// TwinCAT 3 PLC project PLC
// ProgramVersion: 3.1.4024.0
// libraries:
//   Tc2_Standard, * (Beckhoff Automation GmbH)
//   Tc2_System, * (Beckhoff Automation GmbH)
//   Tc3_Module, * (Beckhoff Automation GmbH)
//   VisuSymbols,3.5.10.0,System
// project tree:
//   Counters/ FB2_Counters.TcPOU
//   / GlobalTextList.TcGTLO, GVL.TcGVL, PlcTask.TcTTO, Visualization Manager.TcVMO (not stored)
//   Interface/ DB10_Alias.TcGVL, DIDO.TcGVL, FC10_Alias.TcPOU
//   Main Functie/ DB_PRG1.TcGVL, FC_PRG1.TcPOU
//   POUs/ FC3_Safety.TcPOU, FC_Comms1.TcPOU, FC_Comms2.TcPOU, FC_StartStopReset.TcPOU, MAIN.TcPOU
//   VISUs/ HMI.TcVIS
// real-time tasks:
//   TASK PlcTask: cycle T#10ms, priority 20, ADS port 350
// I/O:
//   DEVICE EC_Master (EtherCAT), AmsNetId 10.10.10.3.2.1
//     Term 1 (EK1100) [EK1100 EtherCAT Coupler (2A E-Bus)]
//       Term 2 (EL1008) [EL1008 8Ch. Dig. Input 24V, 3ms]
//       Term 3 (EL1008) [EL1008 8Ch. Dig. Input 24V, 3ms]
//       Term 4 (EL2004) [EL2004 4Ch. Dig. Output 24V, 0.5A]
//       Term 5 (EL2004) [EL2004 4Ch. Dig. Output 24V, 0.5A]
//       Term 6 (EL2004) [EL2004 4Ch. Dig. Output 24V, 0.5A]
//       Term 7 (EL9011) [EL9011 End Terminal]
// variable links:
//   PLC/PLC Instance <-> EC_Master (EtherCAT)/Term 1 (EK1100)/Term 2 (EL1008)
//     PlcTask Inputs/DIDO.Ingang{1..8} <-> Channel {1..8}/Input  (8 links)
//   PLC/PLC Instance <-> EC_Master (EtherCAT)/Term 1 (EK1100)/Term 3 (EL1008)
//     PlcTask Inputs/DIDO.Ingang{9..16} <-> Channel {1..8}/Input  (8 links)
//   PLC/PLC Instance <-> EC_Master (EtherCAT)/Term 1 (EK1100)/Term 4 (EL2004)
//     PlcTask Outputs/DIDO.Uitgang{1..4} <-> Channel {1..4}/Output  (4 links)
//   PLC/PLC Instance <-> EC_Master (EtherCAT)/Term 1 (EK1100)/Term 5 (EL2004)
//     PlcTask Outputs/DIDO.Uitgang{5..8} <-> Channel {1..4}/Output  (4 links)
//   PLC/PLC Instance <-> EC_Master (EtherCAT)/Term 1 (EK1100)/Term 6 (EL2004)
//     PlcTask Outputs/DIDO.Uitgang{9..12} <-> Channel {1..4}/Output  (4 links)

CONFIGURATION PLC
    RESOURCE PLC ON TwinCAT3
        TASK PlcTask(INTERVAL := T#10ms, PRIORITY := 20);
        PROGRAM MAIN WITH PlcTask : MAIN;
    END_RESOURCE
END_CONFIGURATION

// ---- GVL.TcGVL
{attribute 'qualified_only'}
VAR_GLOBAL
	
	safetyOK : BOOL := FALSE;
	b_StartPRG : BOOL;
	b_StopPRG : BOOL;
	// KUKA communicaties	
	i_KUKAStatus : INT;
	b_startBeweging : BOOL;
END_VAR

// ---- Interface/DB10_Alias.TcGVL
{attribute 'qualified_only'}
VAR_GLOBAL
		

	b_IOSimulatie : BOOL := FALSE;
	// ingangen Nood, start & stop
	ix_E_stopNC : BOOL;
	ix_startKnop : BOOL;
	ix_stopKnop : BOOL; 
	
	// ingangen fotocel
	ix_lengteFC : BOOL;
	ix_hamsterGripperDetectieFC : BOOL;
	
	ix_reedCuttingtoolCilinderOpen : BOOL;
	ix_reedCuttingtoolCilinderGesloten : BOOL;
	ix_reedGripperCilinder1 : BOOL;
	ix_reedGripperCilinder2 : BOOL;
	
	// start/ stop uitgangen extruder&cutting tool
	qx_relaisExtruderStart : BOOL;
	qx_relaisExtruderStop: BOOL;
	qx_relaisCuttingtoolActiveer : BOOL;
	qx_relaisCuttingtoolDeactiveer : BOOL;
	
	// uitgangen ventielaansturing
	qx_ventielEen : BOOL; 
	qx_ventielTwee : BOOL; 
	
	//uitgangen gereserveerd voor KUKA/Engel communicatie
	// E stop
	// bitlevel comm's
	qx_kukaCommEstop : BOOL; 	// E_stop
	qx_kukaCommStart : BOOL; 		// startcommando
	ix_kukaGereed : BOOL; 		// Gereed/persencompleet
	ix_kukaAlarmIN : BOOL; 		// alarm
	
	
END_VAR

// ---- Interface/DIDO.TcGVL
{attribute 'qualified_only'}
VAR_GLOBAL
	

	// Digitale ingangen
	Ingang1 AT %IX40.0 : BOOL;
	Ingang2 AT %IX40.1 : BOOL;
	Ingang3 AT %IX40.2 : BOOL;
	Ingang4 AT %IX40.3 : BOOL;
	Ingang5 AT %IX40.4 : BOOL;
	Ingang6 AT %IX40.5 : BOOL;
	Ingang7 AT %IX40.6 : BOOL;
	Ingang8 AT %IX40.7 : BOOL;

	Ingang9 AT %IX41.0 : BOOL;
	Ingang10 AT %IX41.1 : BOOL;
	Ingang11 AT %IX41.2 : BOOL;
	Ingang12 AT %IX41.3 : BOOL;
	Ingang13 AT %IX41.4 : BOOL;
	Ingang14 AT %IX41.5 : BOOL;
	Ingang15 AT %IX41.6 : BOOL;
	Ingang16 AT %IX41.7 : BOOL;
	
	
	// Digitale uitgangen
	Uitgang1 AT %QX26.0 : BOOL;
	Uitgang2 AT %QX26.1 : BOOL;
	Uitgang3 AT %QX26.2 : BOOL;
	Uitgang4 AT %QX26.3 : BOOL;
	Uitgang5 AT %QX26.4 : BOOL;
	Uitgang6 AT %QX26.5 : BOOL;
	Uitgang7 AT %QX26.6 : BOOL;
	Uitgang8 AT %QX26.7 : BOOL;
	Uitgang9 AT %QX27.0 : BOOL;
	Uitgang10 AT %QX27.1 : BOOL;
	Uitgang11 AT %QX27.2 : BOOL;
	Uitgang12 AT %QX27.3 : BOOL;	
	
END_VAR

// ---- Main Functie/DB_PRG1.TcGVL
{attribute 'qualified_only'}
VAR_GLOBAL
	PRG1Stap : INT;
	
	t_prgT1_extruderRelaisAan : TON;
	t_prgT2_extruderRelaisStop : TON;
	t_prgT3_cuttingRelaisAan : TON;
	t_prgT4_cuttingRelaisUit : TON;
	t_prgT5_resetKukaGereed : TON; // <<<<<<<<<<<<<<<<< Ter simulatie. IRL signaal van KUKA die dit regelt.
	t_prgT6_Stap60advance : TON;
	t_prgT7_PRGStopRelaisTimer : TON;
	t_prgT8 : TON;
END_VAR

// ---- POUs/MAIN.TcPOU
PROGRAM MAIN
VAR
	FB2_Counters : FB2_Counters;

END_VAR

// Init spulletjes

FB2_Counters();
FC10_Alias();

GVL.safetyOK := FC3_Safety();

// FC Comms from KUKA.
GVL.i_KUKAStatus := FC_Comms1(DB10_Alias.ix_kukaGereed,DB10_Alias.ix_kukaAlarmIN);

FC_StartStopReset();

FC_PRG1(GVL.safetyOK, GVL.i_KUKAStatus); // hardcoded '1' vanaf de KUKA; // GVL.i_KUKAStatus

// FC COmms to KUKA
	
FC_Comms2(GVL.safetyOK,GVL.b_startBeweging);

END_PROGRAM

// ---- Counters/FB2_Counters.TcPOU
FUNCTION_BLOCK FB2_Counters
VAR_INPUT
END_VAR
VAR_OUTPUT
END_VAR
VAR
	t_timerHigh : TON;
	t_timerLow : TP;
	b_eenHzClk : BOOL;
	b_eenHzTrigger : R_Trig;
	i_productieTimerSec: DINT;
	i_productieTimerMin: DINT;
	i_productieTimerHour: DINT;
END_VAR
VAR // added by the converter: edge detectors and wires of the graphical bodies
    _w1, _w2 : BOOL;
END_VAR

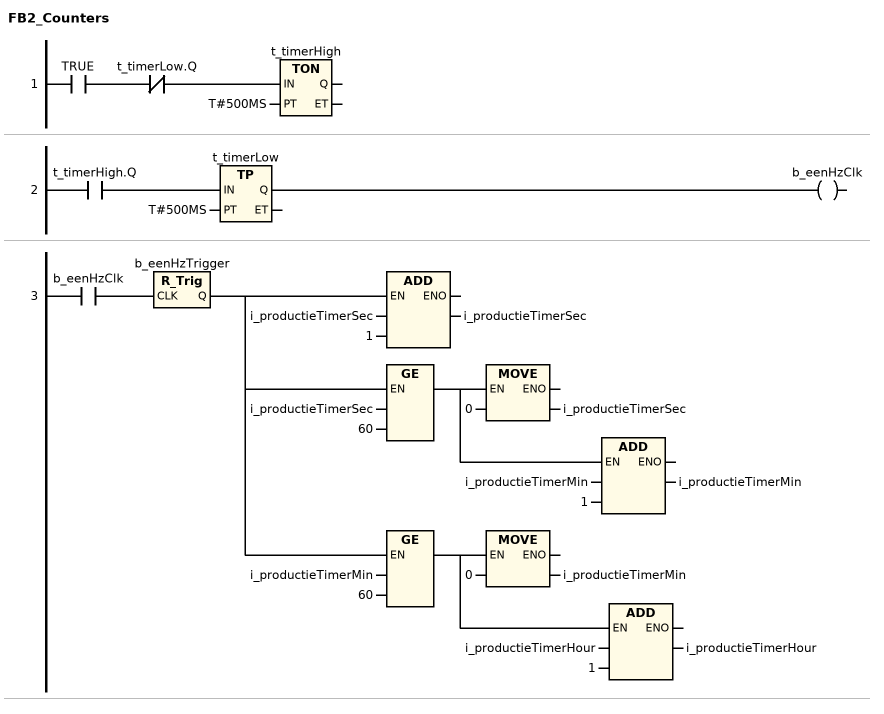
// NETWORK 1
t_timerHigh(IN := TRUE AND NOT t_timerLow.Q, PT := T#500MS); // TON

// NETWORK 2
t_timerLow(IN := t_timerHigh.Q, PT := T#500MS); // TP
b_eenHzClk := t_timerLow.Q;

// NETWORK 3
b_eenHzTrigger(CLK := b_eenHzClk); // R_Trig
IF b_eenHzTrigger.Q THEN i_productieTimerSec := i_productieTimerSec + 1; END_IF
_w1 := b_eenHzTrigger.Q AND i_productieTimerSec >= 60;
IF _w1 THEN i_productieTimerSec := 0; END_IF
IF _w1 THEN i_productieTimerMin := i_productieTimerMin + 1; END_IF
_w2 := b_eenHzTrigger.Q AND i_productieTimerMin >= 60;
IF _w2 THEN i_productieTimerMin := 0; END_IF
IF _w2 THEN i_productieTimerHour := i_productieTimerHour + 1; END_IF

END_FUNCTION_BLOCK

// ---- Interface/FC10_Alias.TcPOU
FUNCTION FC10_Alias : BOOL
VAR_INPUT
END_VAR
VAR
END_VAR

IF NOT DB10_Alias.b_IOSimulatie THEN
		
	// ingangen Noodstop
	DB10_Alias.ix_E_stopNC := DIDO.Ingang15;
	DB10_Alias.ix_startKnop := DIDO.Ingang8;
	DB10_Alias.ix_stopKnop := DIDO.Ingang7; 
	
	// ingangen fotocel
	DB10_Alias.ix_lengteFC := NOT DIDO.Ingang5;
	//DB10_Alias.ix_hamsterGripperDetectieFC := NOT DIDO.Ingang6;
	

	//DB10_Alias.ix_reedCuttingtoolCilinderOpen := DIDO.Ingang13;
	//DB10_Alias.ix_reedCuttingtoolCilinderGesloten := DIDO.Ingang14;
	//DB10_Alias.ix_reedGripperCilinder1 := BOOL;
	//DB10_Alias.ix_reedGripperCilinder2 := BOOL;
	
	// uitgangen - status uit DB10_Alias
	DIDO.Uitgang9 := DB10_Alias.qx_relaisExtruderStart;
	DIDO.Uitgang10 := DB10_Alias.qx_relaisExtruderStop;
	DIDO.Uitgang11 := DB10_Alias.qx_relaisCuttingtoolActiveer;
	DIDO.Uitgang12 := DB10_Alias.qx_relaisCuttingtoolDeactiveer;
	
	// uitgangen ventielaansturing
	DIDO.Uitgang3 := DB10_Alias.qx_ventielEen;
	//DIDO.UitgangX := DB10_Alias.qx_ventielTwee; 
	
	// uitgangen gereserveerd voor KUKA/Engel communicatie
	DIDO.Uitgang7 := DB10_Alias.qx_kukaCommEstop; 	// E_stop
	DIDO.Uitgang8 := DB10_Alias.qx_kukaCommStart; 	// startcommando
	//DB10_Alias.ix_kukaGereed := DIDO.Ingang9; 		// persencompleet
	//DB10_Alias.ix_kukaAlarmIN := DIDO.Ingang10; 	// alarm

END_IF

END_FUNCTION

// ---- POUs/FC3_Safety.TcPOU
FUNCTION FC3_Safety : BOOL
VAR_INPUT
END_VAR
VAR
END_VAR



IF  DB10_Alias.ix_E_stopNC AND NOT DB10_Alias.ix_kukaAlarmIN THEN
	
	FC3_Safety := TRUE;
ELSE
	FC3_Safety := FALSE;
	GVL.b_StopPRG := TRUE;
	DB10_Alias.qx_ventielEen := FALSE;
END_IF

END_FUNCTION

// ---- POUs/FC_Comms1.TcPOU
FUNCTION FC_Comms1 : INT
VAR_INPUT
	ix_gereed : BOOL;
	ix_ALARM : BOOL;
	//ix_bewegingVoltooid : BOOL;
END_VAR
VAR
END_VAR

// KUKA Robot naar PLC communicatie;

IF DB_PRG1.PRG1Stap = 60 AND NOT ix_ALARM THEN		//status beweging actief
	FC_Comms1 := 2;
ELSIF ix_gereed AND NOT ix_ALARM THEN								//status gereed wacht op beweeg
	FC_Comms1 := 1;
ELSIF ix_ALARM THEN													// status alarms
	FC_Comms1 := 4;
ELSE 
	FC_Comms1 := 3;													// iets anders 
END_IF

END_FUNCTION

// ---- POUs/FC_StartStopReset.TcPOU
FUNCTION FC_StartStopReset : BOOL
VAR_INPUT
END_VAR
VAR
END_VAR

// start/stopknop regeling
IF (DB10_Alias.ix_stopKnop AND DB10_Alias.ix_startKnop) OR NOT GVL.safetyOK THEN
	DB_PRG1.PRG1Stap := 950;	 

ELSIF DB10_Alias.ix_stopKnop THEN
	GVL.b_StopPRG := TRUE;
	GVL.b_StartPRG := FALSE;
ELSIF DB10_Alias.ix_startKnop AND GVL.i_KUKAStatus = 1 THEN
	GVL.b_StartPRG := TRUE;
	GVL.b_StopPRG := FALSE;
END_IF
IF GVL.b_StopPRG THEN
	DB_PRG1.PRG1Stap := 900;
END_IF

END_FUNCTION

// ---- Main Functie/FC_PRG1.TcPOU
FUNCTION FC_PRG1 : BOOL
VAR_INPUT
	SafetyOK : BOOL;
	KukaStatus : INT;
END_VAR
VAR

	Foutcode : INT; 
	Melding : STRING[20];
END_VAR




CASE DB_PRG1.PRG1Stap OF
	
	0:
		IF SafetyOK AND KukaStatus = 1 AND GVL.b_StartPRG THEN
			DB_PRG1.PRG1Stap := 5;
		END_IF

	5:
		//extruder start aan
		DB_PRG1.t_prgT1_extruderRelaisAan(IN:=TRUE,PT:=T#2S);
		DB10_Alias.qx_relaisExtruderStart := TRUE;
		
		IF DB_PRG1.t_prgT1_extruderRelaisAan.Q THEN
			DB10_Alias.qx_relaisExtruderStart := FALSE;
			DB_PRG1.t_prgT1_extruderRelaisAan.IN := FALSE;
			DB_PRG1.PRG1Stap := 10;
		END_IF
		
	;
	10: // inlezen fotocel lengte
	
		IF DB10_Alias.ix_lengteFC THEN
			DB_PRG1.PRG1Stap := 20;
		END_IF
		
	
	;
	20: // extruder stop aan bij fotocel
	
		DB10_Alias.qx_relaisExtruderStop := TRUE;
		DB_PRG1.PRG1Stap := 30;
		
	;
	
	30:	// cuttingtool aan en extruderstop laag
		DB10_Alias.qx_relaisCuttingtoolActiveer := TRUE;
		DB_PRG1.t_prgT2_extruderRelaisStop(IN:=TRUE,PT:=T#6S); // 4 seconden timeout voor cuttingtool.
		
		IF DB10_Alias.ix_reedCuttingtoolCilinderGesloten THEN
	
			DB10_Alias.qx_relaisExtruderStop := FALSE;
			DB10_Alias.qx_relaisCuttingtoolActiveer := FALSE;
			DB_PRG1.PRG1Stap:= 40;
		(*ELSIF DB_PRG1.t_prgT2.ET > T#2S THEN
			DB10_Alias.qx_relaisExtruderStop := FALSE;
			DB10_Alias.qx_relaisCuttingtoolActiveer := FALSE;
			DB_PRG1.t_prgT2.IN := FALSE;			*)
		ELSIF DB_PRG1.t_prgT2_extruderRelaisStop.Q THEN
			
			DB_PRG1.t_prgT2_extruderRelaisStop.IN := FALSE;
			Foutcode := 1;
			DB_PRG1.PRG1Stap:= 808;
			
		END_IF
	;
	40:	// cuttingtool deactiveer
		
		DB10_Alias.qx_relaisCuttingtoolDeactiveer := TRUE;	
		DB_PRG1.t_prgT2_extruderRelaisStop.IN := FALSE;
		
		DB_PRG1.t_prgT3_cuttingRelaisAan(IN:=TRUE,PT:=T#6S);
		
		IF DB10_Alias.ix_reedCuttingtoolCilinderOpen THEN
			DB10_Alias.qx_relaisCuttingtoolDeactiveer := FALSE;
			GVL.b_startBeweging := TRUE;
			DB_PRG1.PRG1Stap := 50;
			
		ELSIF DB_PRG1.t_prgT3_cuttingRelaisAan.Q THEN
	
			DB_PRG1.t_prgT3_cuttingRelaisAan.IN := FALSE;
			Foutcode := 2;
			DB_PRG1.PRG1Stap:= 808;
			
		END_IF
	
	50: // Check gripperFC en activeer ventiel.
		IF GVL.i_KUKAStatus = 1 THEN
			
			DB10_Alias.qx_ventielEen := TRUE;
			DB_PRG1.t_prgT5_resetKukaGereed(IN := TRUE,PT:=T#3S);
			DB_PRG1.PRG1Stap := 60;
			
		END_IF
	;
	60:	// Timers zijn ter simulatie. Signalen komen vanaf de KUKA
		DB_PRG1.t_prgT5_resetKukaGereed(IN := TRUE,PT:=T#3S);
		DB_PRG1.t_prgT6_Stap60advance(IN := TRUE,PT:=T#20S);
		IF DB_PRG1.t_prgT5_resetKukaGereed.Q THEN 
			DB_PRG1.t_prgT5_resetKukaGereed(IN := FALSE);
			DB10_Alias.ix_kukaGereed := FALSE; /// <<<<<<<<<<<<<<<<< Ter simulatie. Moet vanaf de Kuka komen.
		END_IF;
		IF DB_PRG1.t_prgT6_Stap60advance.Q AND DB10_Alias.ix_kukaGereed THEN
			DB_PRG1.PRG1Stap := 70;
		END_IF
		
		
		

 
	;
	
	808: // Fout fout hella fout
		
		CASE Foutcode OF
			1: Melding := 'Cuttingtool sluiten fout';
			; 
			2: Melding := 'Cuttingtool openen fout';
			;
			3:
			;
			ELSE
			//DB_PRG1.PRG1Stap := 900;	
			
		END_CASE
			IF GVL.safetyOK THEN
				DB_PRG1.PRG1Stap := 900;
			END_IF 			
	;
	900: // reset en terug naar start.
	
		DB_PRG1.t_prgT7_PRGStopRelaisTimer(IN := TRUE,PT:=T#4S);
		DB10_Alias.qx_relaisCuttingtoolDeactiveer := TRUE;
		DB10_Alias.qx_relaisExtruderStop := TRUE;
		DB10_Alias.qx_ventielEen := FALSE;
		
		IF DB_PRG1.t_prgT7_PRGStopRelaisTimer.Q THEN
			DB10_Alias.qx_relaisCuttingtoolDeactiveer := FALSE;
			DB10_Alias.qx_relaisExtruderStop := FALSE;
			DB_PRG1.t_prgT7_PRGStopRelaisTimer.IN := FALSE;
			DB_PRG1.PRG1Stap := 0;
		END_IF
	;
	
	950: // tussentijdse reset of Safety

		
	;
END_CASE

END_FUNCTION

// ---- POUs/FC_Comms2.TcPOU

FUNCTION FC_Comms2

VAR_INPUT
	ix_Safety : BOOL := FALSE;	
	b_startBeweging : BOOL;
	
END_VAR
VAR
END_VAR
VAR_OUTPUT

END_VAR



DB10_Alias.qx_kukaCommEstop := NOT GVL.safetyOK;
IF DB10_Alias.qx_kukaCommEstop THEN
	DB_PRG1.PRG1Stap := 808;
END_IF
(*
IF DB_PRG1.PRG1Stap = 60 AND NOT DB10_Alias.qx_kukaCommEstop THEN
	DB10_Alias.qx_kukaCommStart := TRUE;
	DB_PRG1.PRG1Stap := 70;
	;
END_IF
*)

END_FUNCTION

// ---- GlobalTextList.TcGTLO
TEXTLIST GlobalTextList
  61 = 'D'
  814 = 'Foutmelding: %i'
  565 = 'Foutmelding: %s'
  520 = 'Gripperventiel'
  522 = 'KUKA Gereed'
  570 = 'KUKA Gereeddicht'
  924 = 'KukaStatus: %i'
  357 = 'Prg Start'
  592 = 'Prg Stop'
  578 = 'PRG1 Stap: %i'
  880 = 'PRG1 Stap: 5i'
  8 = 'PRGStap: %i'
  409 = 'Reed Cilinder dicht'
  700 = 'Reed Cilinder Open'
  71 = 'Reed Cutting Open'
  818 = 'Reed Gripper'
  463 = 'Reed Gripper1'
  124 = 'Safety OK'
  30 = 'Startbeweging'
END_TEXTLIST

// ---- VISUs/HMI.TcVIS
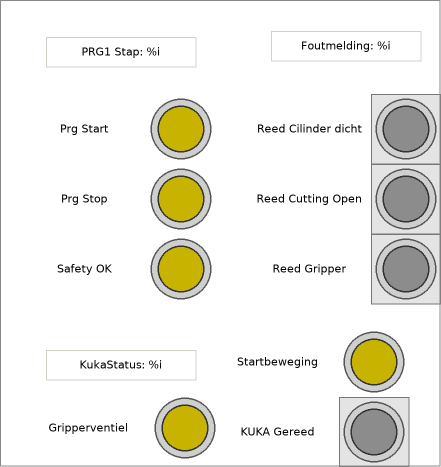
VISUALIZATION HMI  // 441x467
    Group (248,94 193x210)
        PushSwitch (123,0 70x70), variable: DB10_Alias.ix_reedCuttingtoolCilinderGesloten, behaviour: TOGGLE, style: Switch-PushSwitch-Gray
        Label (0,20 123x30), "Reed Cilinder dicht"
        PushSwitch (123,70 70x70), variable: DB10_Alias.ix_reedCuttingtoolCilinderOpen, behaviour: TOGGLE, style: Switch-PushSwitch-Gray
        Label (0,90 123x30), "Reed Cutting Open"
        PushSwitch (123,140 70x70), variable: DB10_Alias.ix_reedGripperCilinder1, behaviour: TAP, style: Switch-PushSwitch-Gray
        Label (0,160 123x30), "Reed Gripper"
    Textfield (46,37 150x30), "PRG1 Stap: %i", text variable: DB_PRG1.PRG1Stap
    Group (23,94 193x70)
        Label (0,20 123x30), "Prg Start"
        Lamp1 (123,0 70x70), variable: GVL.b_StartPRG, style: Lamp-Lamp1-Yellow
    Group (23,164 193x70)
        Label (0,20 123x30), "Prg Stop"
        Lamp1 (123,0 70x70), variable: GVL.b_StopPRG, style: Lamp-Lamp1-Yellow
    Group (23,234 193x70)
        Label (0,20 123x30), "Safety OK"
        Lamp1 (123,0 70x70), variable: GVL.safetyOK, style: Lamp-Lamp1-Yellow
    Textfield (271,31 150x30), "Foutmelding: %i", text variable: FC_PRG1.Foutcode
    Textfield (46,350 150x30), "KukaStatus: %i", text variable: GVL.i_KUKAStatus
    Group (216,327 193x70)
        Label (0,20 123x30), "Startbeweging"
        Lamp1 (123,0 70x70), variable: GVL.b_startBeweging, style: Lamp-Lamp1-Yellow
    PushSwitch (339,397 70x70), variable: DB10_Alias.ix_kukaGereed, behaviour: TOGGLE, style: Switch-PushSwitch-Gray
    Label (216,417 123x30), "KUKA Gereed"
    Label (27,413 123x30), "Gripperventiel"
    Lamp1 (150,393 70x70), variable: DB10_Alias.qx_ventielEen, style: Lamp-Lamp1-Yellow
END_VISUALIZATION
